FUNCTION_BLOCK AutoMode (* Composite Function Block Type *)
  (* Standard: 61499-2 *)
  (* Version 0.0, 2011-12-28, 4DIAC-IDE, 4DIAC-Consortium *)
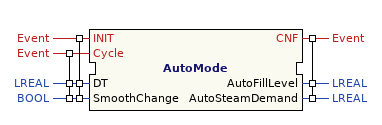
  EVENT_INPUT
    INIT WITH DT, SmoothChange; (* Initialization Request *)
    Cycle WITH DT, SmoothChange;
  END_EVENT
  EVENT_OUTPUT
    CNF WITH AutoFillLevel, AutoSteamDemand; (* Execution Confirmation *)
  END_EVENT
  VAR_INPUT
    DT : LREAL;
    SmoothChange : BOOL := 0;
  END_VAR
  VAR_OUTPUT
    AutoFillLevel : LREAL; (* Output event qualifier *)
    AutoSteamDemand : LREAL;
  END_VAR
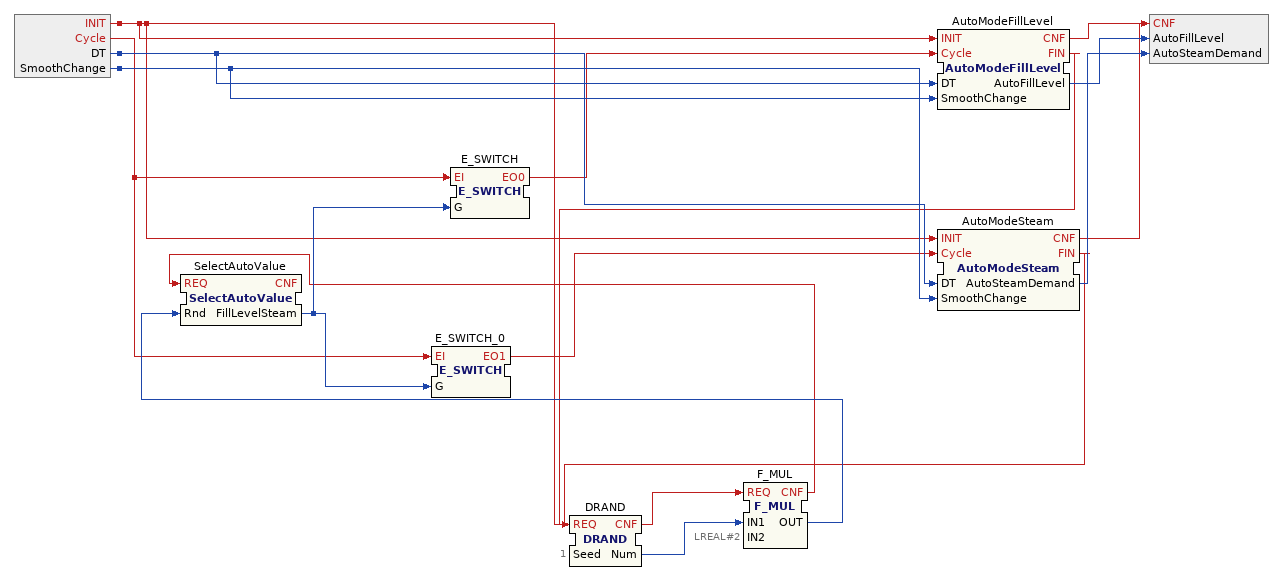
  FBS
    DRAND : DRAND(Seed := 1);
    AutoModeFillLevel : AutoModeFillLevel;
    AutoModeSteam : AutoModeSteam;
    E_SWITCH : E_SWITCH;
    E_SWITCH_0 : E_SWITCH;
    SelectAutoValue : SelectAutoValue;
    F_MUL : F_MUL(IN2 := LREAL#2);
  END_FBS
  EVENT_CONNECTIONS
    AutoModeFillLevel.FIN TO DRAND.REQ;
    AutoModeSteam.FIN TO DRAND.REQ;
    INIT TO AutoModeFillLevel.INIT;
    INIT TO AutoModeSteam.INIT;
    Cycle TO E_SWITCH.EI;
    Cycle TO E_SWITCH_0.EI;
    E_SWITCH.EO0 TO AutoModeFillLevel.Cycle;
    E_SWITCH_0.EO1 TO AutoModeSteam.Cycle;
    INIT TO DRAND.REQ;
    AutoModeFillLevel.CNF TO CNF;
    AutoModeSteam.CNF TO CNF;
    DRAND.CNF TO F_MUL.REQ;
    F_MUL.CNF TO SelectAutoValue.REQ;
  END_CONNECTIONS
  DATA_CONNECTIONS
    DT TO AutoModeFillLevel.DT;
    DT TO AutoModeSteam.DT;
    SmoothChange TO AutoModeFillLevel.SmoothChange;
    SmoothChange TO AutoModeSteam.SmoothChange;
    SelectAutoValue.FillLevelSteam TO E_SWITCH_0.G;
    SelectAutoValue.FillLevelSteam TO E_SWITCH.G;
    AutoModeFillLevel.AutoFillLevel TO AutoFillLevel;
    AutoModeSteam.AutoSteamDemand TO AutoSteamDemand;
    DRAND.Num TO F_MUL.IN1;
    F_MUL.OUT TO SelectAutoValue.Rnd;
  END_CONNECTIONS
END_FUNCTION_BLOCK
